Fanuc KAREL source: kt00058.KL

-- PROVISIONAL review KL for V770-1; original PC SHA256 f01acd149b8da73c53d663fb05c71f2f7056e71b23272c818204580fedc49547
-- Incomplete behavior may be omitted. Consult companion uncertainty JSON. Do not deploy.
PROGRAM KT00058
%NOLOCKGROUP
VAR
  I2 : INTEGER
  OUT : REAL
-- UNRESOLVED_DECL H1 type=002017
BEGIN
  -- UNRESOLVED_PC offsets 5-19; opcodes 2E,22,9D,33,B4
  -- UNRESOLVED_PC offsets 24-35; opcodes 2E,23
  -- UNRESOLVED_PC offsets 40-63; opcodes 22,9D,33,B3,21,53,64,23
  -- UNRESOLVED_PC offsets 68-72; opcodes 7F
END KT00058
